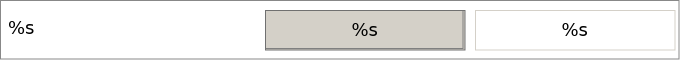
VISUALIZATION SingleRecipesParameterTypeBool  // 680x60
VAR_IN_OUT
	stRecipeParameter : ST_VisuCtrlRecipeParameter;
END_VAR
    Textfield (475,10 200x40), "%s", text variable: stRecipeParameter.sFileValue
    Textfield (5,8 250x40), "%s", text variable: stRecipeParameter.sName
    Button (265,10 200x40), "%s", text variable: stRecipeParameter.sName
        toggle stRecipeParameter.bValue
END_VISUALIZATION

(* stored: Version 1.1.0.1, ProductVersion 3.1.4024.12
   Visu SingleRecipesParameterTypeBool: Id {8c6bd5e0-3a1f-473b-92cb-5080d5209b22} *)
